FUNCTION_BLOCK FB_Cylinder EXTENDS TcNexa_Devices_TcDeviceBase.FB_DeviceBase IMPLEMENTS I_Cylinder
VAR
(*----------------------------------------------------------------------------------------------*)
	sensorHP		AT %I*		: BOOL;
	sensorWP		AT %I*		: BOOL;
	valveHP			AT %Q*		: BOOL;
	valveWP			AT %Q*		: BOOL;
(*----------------------------------------------------------------------------------------------*)
	_inHP						: BOOL;
	_inWP						: BOOL;
	_newStateInterlockHP		: BOOL;
	_newStateInterlockMsgHP		: STRING(255);
	_interlockHP				: BOOL;
	_interlockMessageHP			: STRING(255);
	_newStateInterlockWP		: BOOL;
	_newStateInterlockMsgWP		: STRING(255);
	_interlockWP				: BOOL;
	_interlockMessageWP			: STRING(255);
	_sensorTagHP				: STRING;
	_sensorTagWP				: STRING;
	_monitorMovementTimeout		: BOOL:= TRUE;
	_movementTimeout			: TIME:= T#5S;
	_monitorSensorsOverlap		: BOOL:= TRUE;
	_sensorsOverlapTimeout		: TIME:= T#100MS;
	_notUsedSensorHP			: BOOL;
	_notUsedSensorWP			: BOOL;
	_delayTimeAfterReachedHP	: TIME;
	_delayTimeAfterReachedWP	: TIME;
	_timerTimeout				: Tc2_Standard.TON;
	_timerPositionReached		: Tc2_Standard.TON;
	_timerSensorsOverlap		: Tc2_Standard.TON;
	_timerInHP					: Tc2_Standard.TON;
	_timerInWP					: Tc2_Standard.TON;
(*----------------------------------------------------------------------------------------------*)
END_VAR

METHOD INTERNAL _getErrorMsgPositionNotReached : STRING(255)
VAR_INPUT
	sensor		: STRING;
END_VAR
_getErrorMsgPositionNotReached:= 'Position not reached';
IF (sensor <> '') THEN
	_getErrorMsgPositionNotReached:= Tc2_Standard.CONCAT(STR1:= _getErrorMsgPositionNotReached, STR2:= ' (');
	_getErrorMsgPositionNotReached:= Tc2_Standard.CONCAT(STR1:= _getErrorMsgPositionNotReached, STR2:= sensor);
	_getErrorMsgPositionNotReached:= Tc2_Standard.CONCAT(STR1:= _getErrorMsgPositionNotReached, STR2:= ')');
END_IF
END_METHOD

METHOD INTERNAL _getMsgInterlocked : STRING(255)
VAR_INPUT
END_VAR
_getMsgInterlocked:= Tc2_Standard.CONCAT(STR1:= _nameTag, STR2:= ' interlocked during ');
_getMsgInterlocked:= Tc2_Standard.CONCAT(STR1:= _getMsgInterlocked, STR2:= _calledMethod);
END_METHOD

METHOD INTERNAL _handleInterlocks
VAR_INPUT
END_VAR
_interlockHP:= _newStateInterlockHP;
_interlockMessageHP:= _newStateInterlockMsgHP;
_interlockWP:= _newStateInterlockWP;
_interlockMessageWP:= _newStateInterlockMsgWP;
END_METHOD

METHOD INTERNAL _handlePositionStatus
VAR_INPUT
END_VAR
_timerInHP(
	IN	:= valveHP AND (_notUsedSensorHP OR sensorHP) AND (NOT sensorWP OR NOT _monitorSensorsOverlap),
	PT	:= _delayTimeAfterReachedHP,
	Q	=> _inHP);
_timerInWP(
	IN	:= valveWP AND (_notUsedSensorWP OR sensorWP) AND (NOT sensorHP OR NOT _monitorSensorsOverlap),
	PT	:= _delayTimeAfterReachedWP,
	Q	=> _inWP);
END_METHOD

METHOD PROTECTED _methodHeader : ST_MethodState
VAR_INPUT
	methodName		: Tc2_System.T_MaxString;
END_VAR
IF (_calledMethod = '') THEN
	_calledMethod:= methodName;
	_Step.init();
	_methodTimeout(IN:= FALSE);
	_methodHeader.init:= TRUE;
	_methodHeader.execute:= TRUE;
	_executeMethod:= TRUE;
	_InternalResponse.setBusy(message:= methodName);
ELSIF (_calledMethod = methodName) THEN
	_executeMethod:= TRUE;
	_tmpText:= _getBusyMessage(message:= 'in progress');
	_InternalResponse.setBusy(message:= _tmpText);
	_methodHeader.execute:= TRUE;
ELSE
	_tmpText:= _getBusyMessage(message:= 'in progress');
	_InternalResponse.setBusy(message:= _tmpText);
END_IF
END_METHOD

METHOD addInterlockHP
VAR_INPUT
	condition		: BOOL;
	message			: STRING(255);
END_VAR
IF condition THEN
	_newStateInterlockHP:= TRUE;
	_newStateInterlockMsgHP:= message;
END_IF
END_METHOD

METHOD addInterlockWP
VAR_INPUT
	condition		: BOOL;
	message			: STRING(255);
END_VAR
IF condition THEN
	_newStateInterlockWP:= TRUE;
	_newStateInterlockMsgWP:= message;
END_IF
END_METHOD

PROPERTY delayTimeAfterReachedHP : TIME
GET
delayTimeAfterReachedHP:= _delayTimeAfterReachedHP;
END_GET
SET
_delayTimeAfterReachedHP:= delayTimeAfterReachedHP;
END_SET
END_PROPERTY

PROPERTY delayTimeAfterReachedWP : TIME
GET
delayTimeAfterReachedWP:= _delayTimeAfterReachedWP;
END_GET
SET
_delayTimeAfterReachedWP:= delayTimeAfterReachedWP;
END_SET
END_PROPERTY

METHOD FB_init : BOOL
VAR_INPUT
	bInitRetains 	: BOOL; 	// if TRUE, the retain variables are initialized (warm start / cold start)
	bInCopyCode 	: BOOL;  	// if TRUE, the instance afterwards gets moved into the copy code (online change)
	name			: STRING;
	tag				: STRING;
	sensorTagHP		: STRING;
	sensorTagWP		: STRING;
END_VAR
THIS^._sensorTagHP:= sensorTagHP;
THIS^._sensorTagWP:= sensorTagWP;

_tmpText:= Tc2_Standard.CONCAT(STR1:= 'Interlock - ', STR2:= _nameTag);
_interlockMessageHP:= Tc2_Standard.CONCAT(STR1:= _tmpText, STR2:= '  not in HP');
_interlockMessageWP:= Tc2_Standard.CONCAT(STR1:= _tmpText, STR2:= '  not in WP');
END_METHOD

METHOD PUBLIC FB_main
VAR_INPUT
END_VAR
SUPER^.FB_main();

_handleInterlocks();
_handlePositionStatus();
END_METHOD

METHOD fill
VAR_INPUT
END_VAR
valveHP:= TRUE;
valveWP:= TRUE;
END_METHOD

PROPERTY PUBLIC inHP : BOOL
GET
inHP:= _inHP;
END_GET
END_PROPERTY

PROPERTY interlockMessageHP : STRING(255)
GET
interlockMessageHP:= _interlockMessageHP;
END_GET
END_PROPERTY

PROPERTY interlockMessageWP : STRING(255)
GET
interlockMessageWP:= _interlockMessageWP;
END_GET
END_PROPERTY

PROPERTY PUBLIC inWP : BOOL
GET
inWP:= _inWP;
END_GET
END_PROPERTY

PROPERTY monitorMovementTimeout : BOOL
GET
monitorMovementTimeout:= _monitorMovementTimeout;
END_GET
SET
_monitorMovementTimeout:= monitorMovementTimeout;
END_SET
END_PROPERTY

PROPERTY monitorSensorsOverlap : BOOL
GET
monitorSensorsOverlap:= _monitorSensorsOverlap;
END_GET
SET
_monitorSensorsOverlap:= monitorSensorsOverlap;
END_SET
END_PROPERTY

PROPERTY movementTimeout : TIME
GET
movementTimeout:= _movementTimeout;
END_GET
SET
_movementTimeout:= movementTimeout;
END_SET
END_PROPERTY

METHOD PUBLIC moveToHP
VAR_INPUT
	Response		: REFERENCE TO TcNexa_Components_TcProcess.FB_MethodResponse;
END_VAR
_methodState:= _methodHeader(methodName:= 'moving to HP');
				
IF _methodState.init THEN
	_timerTimeout(IN:= FALSE);
	_timerPositionReached(IN:= FALSE);
END_IF

IF _methodState.execute THEN
	IF NOT _interlockHP THEN
		valveHP:= TRUE;
		valveWP:= FALSE;		
		
		_timerTimeout(
			IN:= _monitorMovementTimeout,
			PT:= _movementTimeout);
		_timerPositionReached(
			IN:= (_notUsedSensorHP OR sensorHP) AND (NOT sensorWP OR NOT _monitorSensorsOverlap),
			PT:= _delayTimeAfterReachedHP);
		_timerSensorsOverlap(
			IN:= _monitorSensorsOverlap AND sensorHP AND sensorWP,
			PT:= _sensorsOverlapTimeout);
		(* Error - both sensors active *)
		IF _timerSensorsOverlap.Q THEN
			_InternalResponse.setFail(message:= _getErrorMessage(), description:= 'Both sensors active');
		(* Error movement - end position not reached *)		
		ELSIF _timerTimeout.Q THEN
			_InternalResponse.setFail(message:= _getErrorMessage(), description:= _getErrorMsgPositionNotReached(_sensorTagHP));
		(* Succes - end position reached *)
		ELSIF _timerPositionReached.Q THEN
			_InternalResponse.setPass();
		END_IF
	ELSE
		_InternalResponse.setBusy(message:= _getMsgInterlocked());
		_timerTimeout(IN:= FALSE);
		_timerPositionReached(IN:= FALSE);
	END_IF
END_IF

_methodFooter(Response:= Response);
END_METHOD

METHOD PUBLIC moveToWP
VAR_INPUT
	Response		: REFERENCE TO TcNexa_Components_TcProcess.FB_MethodResponse;
END_VAR
_methodState:= _methodHeader(methodName:= 'moving to WP');
				
IF _methodState.init THEN
	_timerTimeout(IN:= FALSE);
	_timerPositionReached(IN:= FALSE);
END_IF

IF _methodState.execute THEN
	IF NOT _interlockWP THEN
		valveHP:= FALSE;
		valveWP:= TRUE;		
		
		_timerTimeout(
			IN:= _monitorMovementTimeout,
			PT:= _movementTimeout);	
		_timerPositionReached(
			IN:= (_notUsedSensorWP OR sensorWP) AND (NOT sensorHP OR NOT _monitorSensorsOverlap),
			PT:= _delayTimeAfterReachedWP);
		_timerSensorsOverlap(
			IN:= _monitorSensorsOverlap AND sensorHP AND sensorWP,
			PT:= _sensorsOverlapTimeout);
		(* Error - both sensors active *)
		IF _timerSensorsOverlap.Q THEN
			_InternalResponse.setFail(message:= _getErrorMessage(), description:= 'Both sensors active');
		(* Error movement - end position not reached *)		
		ELSIF _timerTimeout.Q THEN
			_InternalResponse.setFail(message:= _getErrorMessage(), description:= _getErrorMsgPositionNotReached(_sensorTagWP));
		(* Succes - end position reached *)
		ELSIF _timerPositionReached.Q THEN
			_InternalResponse.setPass();
		END_IF	
	ELSE
		_InternalResponse.setBusy(message:= _getMsgInterlocked());
		_timerTimeout(IN:= FALSE);
		_timerPositionReached(IN:= FALSE);			
	END_IF
END_IF

_methodFooter(Response:= Response);
END_METHOD

PROPERTY notUsedSensorHP : BOOL
GET
notUsedSensorHP:= _notUsedSensorHP;
END_GET
SET
_notUsedSensorHP:= notUsedSensorHP;
END_SET
END_PROPERTY

PROPERTY notUsedSensorWP : BOOL
GET
notUsedSensorWP:= _notUsedSensorWP;
END_GET
SET
_notUsedSensorWP:= notUsedSensorWP;
END_SET
END_PROPERTY

METHOD PUBLIC off
VAR_INPUT
END_VAR
valveHP:= FALSE;
valveWP:= FALSE;
END_METHOD

PROPERTY sensorsOverlapTimeout : TIME
GET
sensorsOverlapTimeout:= _sensorsOverlapTimeout;
END_GET
SET
_sensorsOverlapTimeout:= sensorsOverlapTimeout;
END_SET
END_PROPERTY

END_FUNCTION_BLOCK

(* stored: Version 1.1.0.1, ProductVersion 3.1.4024.12
   POU FB_Cylinder: Id {680c2ba4-8397-462a-87a8-fe203f1c0cf9}, SpecialFunc None
   Folder Internal: Id {bb5dbec5-7b9a-4878-b8f2-219e5006a525}
   Folder Property: Id {fa0b090e-3187-4873-bac4-b031a80348e4}
   Method _getErrorMsgPositionNotReached: Id {36362996-0261-40b0-8789-ce85c53c967e}
   Method _getMsgInterlocked: Id {9ef63f04-0574-08b4-25d4-13a7b30758b7}
   Method _handleInterlocks: Id {4684f171-6db4-054d-2f96-856891069c62}
   Method _handlePositionStatus: Id {52787e74-8e74-0d86-0e07-7d2e53fe0eb1}
   Method _methodHeader: Id {697a6e2d-5c00-4306-aac2-c0c90b1d5589}
   Method addInterlockHP: Id {ad3bdc61-5cb8-033b-1e59-6dedd0ef52c2}
   Method addInterlockWP: Id {086a0259-2b9d-0334-2432-a78863027101}
   Property delayTimeAfterReachedHP: Id {8c1f2677-0daa-0c05-15ec-88d15dc725ab}
   Get Get: Id {89d296ae-b3a4-0097-1fc9-7850713d38b8}
   Set Set: Id {40cefdc7-3876-05c7-37fe-845da8d79903}
   Property delayTimeAfterReachedWP: Id {2585a8d9-041c-0e7f-3e21-41bee3c91027}
   Get Get: Id {8fc230f5-ecaf-0baf-306f-2432bedd8172}
   Set Set: Id {6682eed0-0ab3-0016-07f8-4bfd82eaaa5d}
   Method FB_init: Id {adaa3848-5907-46de-9004-d792f2e55d84}
   Method FB_main: Id {2dacd2a9-ec5f-0618-3c0a-8ce5c4389064}
   Method fill: Id {65a9eca6-4fe0-0f43-1b39-3aaf0673fea5}
   Property inHP: Id {d3396af4-179b-4b3f-bfb6-638a6f9684d0}
   Get Get: Id {6c32fa55-1d59-473e-864b-6cc4b5cf7c54}
   Property interlockMessageHP: Id {38f74a37-690f-0b2c-3988-cd0be520935e}
   Get Get: Id {2ab42182-b181-0ed9-3c98-ac94fe5e55c6}
   Property interlockMessageWP: Id {73b1be68-b97c-03d8-2c32-42db0d213a42}
   Get Get: Id {99159a4b-3f50-0de6-03a9-e9eecf9304ad}
   Property inWP: Id {34504795-4af5-46fb-acaa-5ed3ea1f163a}
   Get Get: Id {a70c5244-bba8-4f01-9b4a-c3b2b3323977}
   Property monitorMovementTimeout: Id {178637e8-f853-09f4-1497-b8454b30de69}
   Get Get: Id {7de491a8-fc2f-0d0e-0fe3-2810d5cf428f}
   Set Set: Id {5c7e436f-74fc-051b-0cdd-bcac949821ee}
   Property monitorSensorsOverlap: Id {0d4e1ab8-96f8-09ca-140d-8db7e3f8aece}
   Get Get: Id {566caacd-119b-0530-1f3a-cc4866738c24}
   Set Set: Id {98ed81e7-68fa-077e-1917-2d8c2a01a98d}
   Property movementTimeout: Id {85797ff6-b1cd-0b70-1b12-09fbe1fa6efe}
   Get Get: Id {d2c43be1-6279-01b4-078d-29054a2987ac}
   Set Set: Id {030b1093-d0c7-0fb1-3982-feab179c64f1}
   Method moveToHP: Id {21c945cc-2bad-44c0-b6d4-d1a325440fb0}
   Method moveToWP: Id {a67ab8a1-e9d4-4ef6-b3df-9ec2a68ebb19}
   Property notUsedSensorHP: Id {2d4f51c9-129d-01ef-0f57-0cec22e0b974}
   Get Get: Id {15d7e984-af42-0510-0639-aaf0f8cd3499}
   Set Set: Id {90440987-ac58-05b3-3d4d-9c84c218b34b}
   Property notUsedSensorWP: Id {64f7dc39-9329-0fe1-3c0f-b4a2b42462ce}
   Get Get: Id {b5029a0e-bd00-0567-0427-8a01bad6a0b1}
   Set Set: Id {c92be4bc-be71-076b-09b7-f43ecd728d35}
   Method off: Id {039fc145-b972-4f45-8abb-ceb005690470}
   Property sensorsOverlapTimeout: Id {c2d78593-82b3-065f-0242-8309f008178a}
   Get Get: Id {1eb7ea26-eadf-0e53-2e0e-38566a201b00}
   Set Set: Id {4b94f6b5-4dd3-0a13-07d5-b98ef402f9f9} *)
